TYPE Udt_CM_Actuator2State_V2 :
STRUCT
	PI_MANUAL :BOOL;
	PI_AUTO : BOOL;
	PI_HMI_HAND : BOOL;
	
	PI_AlarmHigh_Enable : BOOL;
	PI_AlarmLow_Enable : BOOL;
	
	PI_Alarm_Condition_H : BOOL;
	PI_Alarm_Condition_L : BOOL;
	
	PI_AlarmDelay_H : LREAL;
	PI_AlarmDelay_L : LREAL;
	
	PI_Alarm_Ack_H : BOOL;
	PI_Alarm_Ack_L : BOOL;
	
	PI_Interlock : BOOL;
	(*PO_Interlocked : BOOL;
	
	PO_ALARM_H : BOOL;
	PO_ALARM_L : BOOL;
	
	PO_HMI_HAND_ON: BOOL;
	PO_AUTO_ON : BOOL;
	PO_MANUAL_ON : BOOL;
	PO_ON : BOOL;
	PO_OFF :BOOL;
	*)
	
	PO_MODE : ENUM_MODE_HANDLER;
	
END_STRUCT
END_TYPE

(* stored: Version 1.1.0.1, ProductVersion 3.1.4024.13
   DUT Udt_CM_Actuator2State_V2: Id {7cfb36b3-d937-4193-946d-600e9b3f4e31} *)
